(* IEC 61131-3 sources: InfiniteStateMachine/st/project/library_information, 2 files *)

(* ---- getlibversionnumber-GetLibVersionNumber.st ---- *)
(* --- Interface --- *)
// This function has been automatically generated from the project information.
FUNCTION GetLibVersionNumber : DWORD
VAR_INPUT

END_VAR

(* --- Implementation --- *)
GetLibVersionNumber := 65793;

(* ---- islibreleased-IsLibReleased.st ---- *)
(* --- Interface --- *)
// This function has been automatically generated from the project information.
FUNCTION IsLibReleased : BOOL
VAR_INPUT

END_VAR

(* --- Implementation --- *)
IsLibReleased := FALSE;
